Fanuc KAREL source: compact_preamble.KL

PROGRAM KE00004
%NOLOCKGROUP
%ENVIRONMENT REGOPE
VAR
I:INTEGER;S : STRING[80];STATUS:INTEGER
BEGIN
I=1
S='TEST'
SET_REG_CMT(I,S,STATUS)
END KE00004
